FUNCTION_BLOCK SENSOR
VAR_INPUT
//<!-- PRESPECTIVE_AUTO_INJECT_INPUT_START -->
iActive : BOOL:= False; //Light active
iIntensity : REAL:= 0.75; //Light intensity
//<!-- PRESPECTIVE_AUTO_INJECT_INPUT_END -->
END_VAR
VAR_OUTPUT
//<!-- PRESPECTIVE_AUTO_INJECT_OUTPUT_START -->
oActive : BOOL:= False; //Light active
oIntensity : REAL:= 1; //Light intensity
//<!-- PRESPECTIVE_AUTO_INJECT_OUTPUT_END -->
END_VAR
VAR
//<!-- PRESPECTIVE_AUTO_INJECT_VAR_START -->
//<!-- PRESPECTIVE_AUTO_INJECT_VAR_END -->
END_VAR

END_FUNCTION_BLOCK

(* stored: Version 1.1.0.1, ProductVersion 3.1.4020.6
   POU SENSOR: SpecialFunc None *)
